{attribute addProperty BoxType "EL1512-0000-0017"}
{attribute addProperty Id "StatusAT %I*Status_D97632771620Counter_valueAT %I*UDINT32417"}
{attribute addProperty CRC "3588638702"}
{attribute addProperty SizeInBites "48"}
{attribute addProperty SizeInBytes "6"}
TYPE CNT_Inputs_Channel_D5E647EE :
STRUCT
	{attribute addProperty Name "Status"}
	Status AT %I* : Status_D9763277;
	{attribute addProperty Name "Counter_value"}
	Counter_value AT %I* : UDINT;
END_STRUCT
END_TYPE

(* stored: Version 1.2.0.0, ProductVersion 3.1.4024.9
   DUT CNT_Inputs_Channel_D5E647EE: Id {96fea424-550a-4347-9a7d-0bf74827d419} *)
